{attribute 'qualified_only'}
{attribute 'strict'}

{attribute 'BaParam.Enum.eAdd.DE' := 'Hinzufügen'}
{attribute 'BaParam.Enum.eAdd.EN' := 'Add'}
{attribute 'BaParam.Enum.eSubstract.DE' := 'Abziehen'}
{attribute 'BaParam.Enum.eSubstract.EN' := 'Substract'}
TYPE E_UDef_Mode :
(
	eAdd,
	eSubstract
);
END_TYPE

(* stored: Version 1.1.0.1, ProductVersion 3.1.4024.9
   DUT E_UDef_Mode: Id {1581ea81-64b9-4594-ba41-d67828c9efc1} *)
